GLOBALCONSTANTS DefaultPool_Numeric (* Numeric object pool constants (ID, Scale, Offset, Decimals) *)
  PACKAGE FBs::Counter::const;
  VAR_GLOBAL CONSTANT
    InputNumber_Gesamtziel : logiBUS::utils::conversion::phys::NumericObjectPool_S := (u16ObjId := 9000, r32Scale := 1.0, i32Offset := 0, u8Decimals := 0);
    InputNumber_Tagesziel : logiBUS::utils::conversion::phys::NumericObjectPool_S := (u16ObjId := 9001, r32Scale := 1.0, i32Offset := 0, u8Decimals := 0);
    OutputNumber_Tageszaehler : logiBUS::utils::conversion::phys::NumericObjectPool_S := (u16ObjId := 12000, r32Scale := 1.0, i32Offset := 0, u8Decimals := 0);
    OutputNumber_Gesamtzaehler : logiBUS::utils::conversion::phys::NumericObjectPool_S := (u16ObjId := 12003, r32Scale := 1.0, i32Offset := 0, u8Decimals := 0);
    NumberVariable_Tageszaehler : logiBUS::utils::conversion::phys::NumericObjectPool_S := (u16ObjId := 21000, r32Scale := 1.0, i32Offset := 0, u8Decimals := 0);
    NumberVariable_Gesamtzaehler : logiBUS::utils::conversion::phys::NumericObjectPool_S := (u16ObjId := 21001, r32Scale := 1.0, i32Offset := 0, u8Decimals := 0);
    NumberVariable_Gesamtziel : logiBUS::utils::conversion::phys::NumericObjectPool_S := (u16ObjId := 21002, r32Scale := 1.0, i32Offset := 0, u8Decimals := 0);
    NumberVariable_Tagesziel : logiBUS::utils::conversion::phys::NumericObjectPool_S := (u16ObjId := 21003, r32Scale := 1.0, i32Offset := 0, u8Decimals := 0);
  END_VAR
END_GLOBALCONSTANTS
